PROGRAM AUTO_POSITION
VAR
END_VAR

END_PROGRAM

(* stored: Version 1.1.0.1, ProductVersion 3.1.4022.18
   POU AUTO_POSITION: Id {cdfbe012-5152-443d-959b-b56c2dafcd18}, SpecialFunc None *)
